FUNCTION_BLOCK PLOT_JSON_TIMESERIES
  {SET_ATTRIBUTE(OpcUa, SERVICE)}
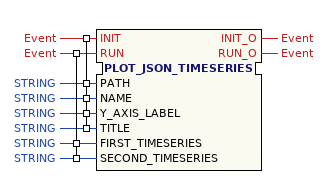
  EVENT_INPUT
    INIT WITH PATH, NAME, Y_AXIS_LABEL, TITLE;
    RUN WITH FIRST_TIMESERIES, SECOND_TIMESERIES;
  END_EVENT
  EVENT_OUTPUT
    INIT_O;
    RUN_O;
  END_EVENT
  VAR_INPUT
    PATH : STRING; {SET_ATTRIBUTE(OpcUa, Constant.RUN)}
    NAME : STRING; {SET_ATTRIBUTE(OpcUa, Constant.RUN)}
    Y_AXIS_LABEL : STRING; {SET_ATTRIBUTE(OpcUa, Constant.RUN)}
    TITLE : STRING; {SET_ATTRIBUTE(OpcUa, Constant.RUN)}
    FIRST_TIMESERIES : STRING; {SET_ATTRIBUTE(OpcUa, Variable.RUN)}
    SECOND_TIMESERIES : STRING; {SET_ATTRIBUTE(OpcUa, Variable.RUN)}
  END_VAR
END_FUNCTION_BLOCK
